PROGRAM ElevatorTask
VAR
	//Varibles booleans
	bAllPrepared 		: BOOL;
	bPressButton 		: BOOL;
	bElevatorArrives 	: BOOL;
	bEnterElevator 		: BOOL;
	bPressFirstFloor	: BOOL;
	bCheckClass 		: BOOL;
	bGoToUniversity 	: BOOL;
	bGoToGym			: BOOL;
	bDone				: BOOL;
	//Variables timers	
	fbGoToElevator 		: TON;
	fbWaitElevator 		: TON;
	fbGoToFirstFloor 	: TON;
	fbWalkToUniversity	: TON;
	fbWalkToClassroom	: TON;
END_VAR

//First step: When i finish my breakfast i prepare my thing and go to take the elevator
	IF GVL.bReady THEN
		bAllPrepared := TRUE;
		fbGoToElevator(IN:=bAllPrepared,PT:=T#3S);
	END_IF

	IF fbGoToElevator.Q THEN
		bPressButton := TRUE;
		fbWaitElevator(IN:=bPressButton,PT:=T#3S);
	END_IF
	
	IF fbWaitElevator.Q THEN
		bElevatorArrives := TRUE;
		bEnterElevator :=bElevatorArrives;
		bPressFirstFloor := bEnterElevator;
		fbGoToFirstFloor(IN:=bPressFirstFloor,PT:=T#4S);
	END_IF
//Second step: When im in the first floor i decide where i want to go

	bCheckClass := ElevatorFunction(bCheckClass := fbGoToFirstFloor.Q);		//Function
	
	IF bCheckClass THEN
		bGoToUniversity := TRUE;
		bGoToGym := FALSE;
	ELSE
		bGoToUniversity := FALSE;
		bGoToGym := TRUE;
	END_IF

//Third step: Go to university and classroom

	fbWalkToUniversity(IN:=bGoToUniversity,PT:=T#5S);
	fbWalkToClassroom(IN:=fbWalkToUniversity.Q,PT:=T#5S);
	
	bDone := fbWalkToClassroom.Q;											//Me in classroom

END_PROGRAM

(* stored: Version 1.1.0.1, ProductVersion 3.1.4024.12
   POU ElevatorTask: Id {f124a62b-2626-46c8-805b-bc427e24398b}, SpecialFunc None *)
